# EPICS substitutions: iocBoot/iocTomoScan_prisma/tomoScan.substitutions
file "$(TOP)/db/tomoScan.template"
{
pattern
{  P,      R,      CAMERA,    FILE_PLUGIN,   ROTATION,  SAMPLE_X,  SAMPLE_Y,      CLOSE_SHUTTER,        CLOSE_VALUE,        OPEN_SHUTTER,         OPEN_VALUE}
{pxm1:, TomoScan:, SIM1:,   SIM1:HDF1:,  spxm1:m1,   SMC01:D,  SMC01:E,        mk4:KvOn,                0,                  mk4:KvOn,      1}
}

file "$(TOP)/tomoScanApp/Db/tomoScan_prisma.template"
{
pattern
{  P,      R}
{pxm1:, TomoScan:}
}
